{attribute 'qualified_only'}
{attribute 'strict'}
{attribute 'to_string'}
TYPE E_UsbLicenseDongleSate : // for (C9900-L100 License-Key-USB-Stick) > BoxInfo > BoxStateVar
(
	NO_ERROR			:= 16#0000,	// 0x0000 = No error
	NO_ACTUAL_INPUTS	:= 16#0001,	// 0x0001 = No actual inputs
	NOT_FOUND			:= 16#0004	// 0x0004 = Not found
) UINT:=NOT_FOUND; // this will be overwritten by Real Dongle State
END_TYPE

(* stored: Version 1.1.0.1, ProductVersion 3.1.4026.20
   DUT E_UsbLicenseDongleSate: Id {e1fc66c9-f12b-4f1d-bd34-656134e80299} *)
